// Mitsubishi GX Works2 project: PLC 특수기능 (Flip Flop 내부 구조)   PLC: Q03UDV

PROGRAM MAIN
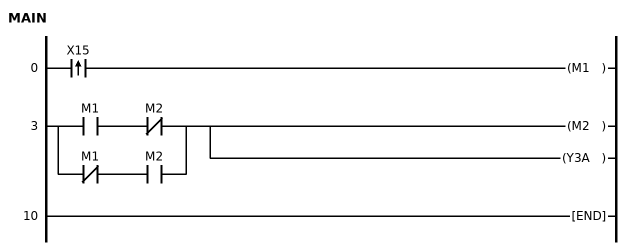
0     LDP     X15
      OUT     M1
3     LD      M1
      ANI     M2
      LDI     M1
      AND     M2
      ORB
      OUT     M2
      OUT     Y3A
10    END
END_PROGRAM
